INTERFACE I_PtTimesource

METHOD getDateTime : PtDateTime
VAR_INPUT
END_VAR
END_METHOD

END_INTERFACE

(* stored: Version 1.1.0.1, ProductVersion 3.1.4024.12
   Itf I_PtTimesource: Id {94cbb150-aaca-4bc5-82c2-1ae2c32b0807}
   Method getDateTime: Id {c44caa02-c7ef-47e3-8b3c-3536d88ee987} *)
